{attribute addProperty BoxType "EJ5151-0000-0016"}
{attribute addProperty Id "ControlAT %Q*Control_38B054C81621Set_counter_valueAT %Q*UINT16217"}
{attribute addProperty CRC "57679667"}
{attribute addProperty SizeInBites "32"}
{attribute addProperty SizeInBytes "4"}
TYPE ENC_Outputs_03701F33 :
STRUCT
	{attribute addProperty Name "Control"}
	Control AT %Q* : Control_38B054C8;
	{attribute addProperty Name "Set_counter_value"}
	Set_counter_value AT %Q* : UINT;
END_STRUCT
END_TYPE

(* stored: Version 1.2.0.0, ProductVersion 3.1.4024.9
   DUT ENC_Outputs_03701F33: Id {378b9ae2-3693-4e24-a1dd-a8ec55eb7eb9} *)
